FUNCTION_BLOCK M2DoThermalFocusForStationName EXTENDS BaseProcess
VAR_INPUT
	///Arguments to be set, before writing do_request TRUE
	{attribute 'OPC.UA.DA' := '1'}
	set: M2DoThermalFocusForStationNameArgs;
END_VAR
VAR_OUTPUT
	///Arguments in use by the process, if do_request was accepted
	{attribute 'OPC.UA.DA' := '1'}
	{attribute 'OPC.UA.DA.Access' := '1'}
	get: M2DoThermalFocusForStationNameArgs;
END_VAR
VAR_IN_OUT
END_VAR
VAR
END_VAR

IF do_request THEN
    do_request_result := request( station := set.station );
    do_request := FALSE;
END_IF;
SUPER^();

{attribute 'TcRpcEnable' := '1'}
METHOD request : RequestResults
VAR_INPUT
	///The configured station name, for which the thermal focus should be executed
	station: STRING;
END_VAR
VAR_OUTPUT
END_VAR
VAR_IN_OUT
END_VAR
VAR
END_VAR
IF THIS^.statuses.enabledStatus.enabled THEN
    THIS^.start( station := station );
    request := RequestResults.ACCEPTED;
ELSE
    request := RequestResults.REJECTED;
END_IF;
END_METHOD

{attribute 'TcRpcEnable' := '1'}
METHOD start
VAR_INPUT
	///The configured station name, for which the thermal focus should be executed
	station: STRING;
END_VAR
VAR_OUTPUT
END_VAR
VAR_IN_OUT
END_VAR
VAR
END_VAR
THIS^.get.station := station;
THIS^.statuses.busyStatus( isBusy := TRUE );
THIS^.statuses.healthStatus( isGood := TRUE );
END_METHOD

END_FUNCTION_BLOCK

(* stored: Version 1.1.0.1, ProductVersion 3.1.4019.2
   POU M2DoThermalFocusForStationName: Id {ec4abfa2-5055-4074-a861-f172b7a936f6}, SpecialFunc None
   Method request: Id {5b9c40ee-15f9-41d4-87a6-a4125cf2eb0e}
   Method start: Id {f3052df2-487f-4066-ade7-88a1351a671f} *)
